% RSLogix 500 project INTRO TO PLC JOB 23 GREG.RSS, saved by version 10.00.00.00 %
PROJECT "UNTITLED"    % processor: Bul.1763 MicroLogix 1100 Series B %

PROGRAM FILES
  LAD 2   25 rungs

DATA FILES
  O0 OUTPUT  4 elements
  I1 INPUT  6 elements
  S2 STATUS  66 elements
  B3 BINARY  1 elements
  T4 TIMER  5 elements
  C5 COUNTER  8 elements
  R6 CONTROL  1 elements
  N7 INTEGER  1 elements
  F8 FLOAT  1 elements

LADDER 2
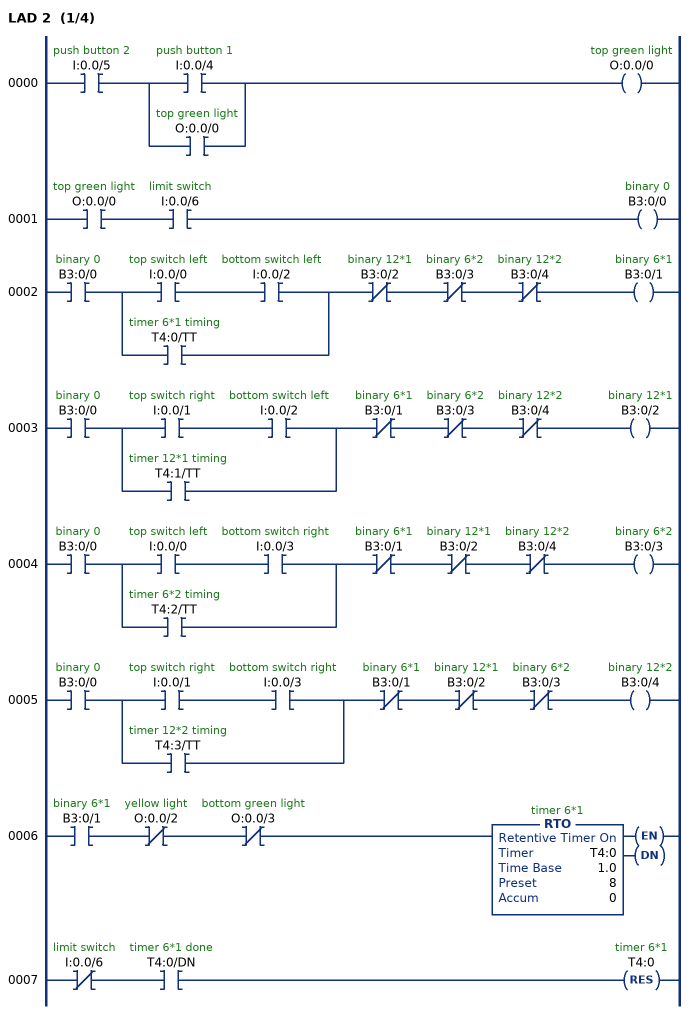
% Rung: 0 %
SOR XIC I:0.0/5 BST XIC I:0.0/4 NXB XIC O:0.0/0 BND OTE O:0.0/0 EOR
%   I:0.0/5  "push button 2" %
%   I:0.0/4  "push button 1" %
%   O:0.0/0  "top green light" %
% Rung: 1 %
SOR XIC O:0.0/0 XIC I:0.0/6 OTE B3:0/0 EOR
%   O:0.0/0  "top green light" %
%   I:0.0/6  "limit switch" %
%   B3:0/0  "binary 0" %
% Rung: 2 %
SOR XIC B3:0/0 BST XIC I:0.0/0 XIC I:0.0/2 NXB XIC T4:0/TT BND XIO B3:0/2 XIO B3:0/3 XIO B3:0/4 OTE B3:0/1 EOR
%   B3:0/0  "binary 0" %
%   I:0.0/0  "top switch left" %
%   I:0.0/2  "bottom switch left" %
%   T4:0/TT  "timer 6*1 timing" %
%   B3:0/2  "binary 12*1" %
%   B3:0/3  "binary 6*2" %
%   B3:0/4  "binary 12*2" %
%   B3:0/1  "binary 6*1" %
% Rung: 3 %
SOR XIC B3:0/0 BST XIC I:0.0/1 XIC I:0.0/2 NXB XIC T4:1/TT BND XIO B3:0/1 XIO B3:0/3 XIO B3:0/4 OTE B3:0/2 EOR
%   B3:0/0  "binary 0" %
%   I:0.0/1  "top switch right" %
%   I:0.0/2  "bottom switch left" %
%   T4:1/TT  "timer 12*1 timing" %
%   B3:0/1  "binary 6*1" %
%   B3:0/3  "binary 6*2" %
%   B3:0/4  "binary 12*2" %
%   B3:0/2  "binary 12*1" %
% Rung: 4 %
SOR XIC B3:0/0 BST XIC I:0.0/0 XIC I:0.0/3 NXB XIC T4:2/TT BND XIO B3:0/1 XIO B3:0/2 XIO B3:0/4 OTE B3:0/3 EOR
%   B3:0/0  "binary 0" %
%   I:0.0/0  "top switch left" %
%   I:0.0/3  "bottom switch right" %
%   T4:2/TT  "timer 6*2 timing" %
%   B3:0/1  "binary 6*1" %
%   B3:0/2  "binary 12*1" %
%   B3:0/4  "binary 12*2" %
%   B3:0/3  "binary 6*2" %
% Rung: 5 %
SOR XIC B3:0/0 BST XIC I:0.0/1 XIC I:0.0/3 NXB XIC T4:3/TT BND XIO B3:0/1 XIO B3:0/2 XIO B3:0/3 OTE B3:0/4 EOR
%   B3:0/0  "binary 0" %
%   I:0.0/1  "top switch right" %
%   I:0.0/3  "bottom switch right" %
%   T4:3/TT  "timer 12*2 timing" %
%   B3:0/1  "binary 6*1" %
%   B3:0/2  "binary 12*1" %
%   B3:0/3  "binary 6*2" %
%   B3:0/4  "binary 12*2" %
% Rung: 6 %
SOR XIC B3:0/1 XIO O:0.0/2 XIO O:0.0/3 RTO T4:0 1.0 8 0 EOR
%   B3:0/1  "binary 6*1" %
%   O:0.0/2  "yellow light" %
%   O:0.0/3  "bottom green light" %
%   T4:0  "timer 6*1" %
% Rung: 7 %
SOR XIO I:0.0/6 XIC T4:0/DN RES T4:0 EOR
%   I:0.0/6  "limit switch" %
%   T4:0/DN  "timer 6*1 done" %
%   T4:0  "timer 6*1" %

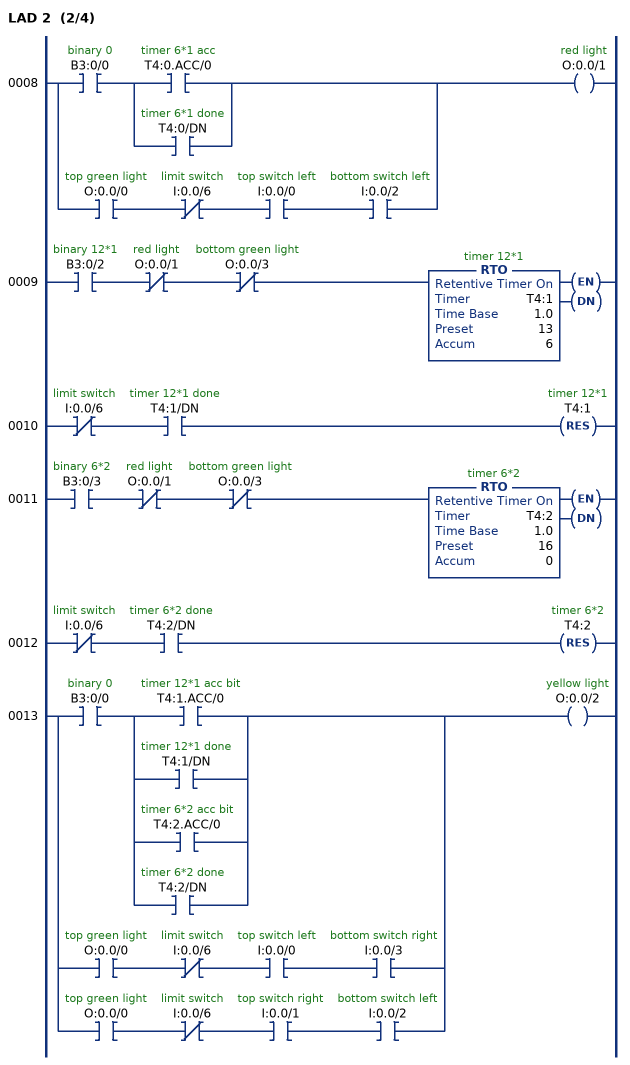
% Rung: 8 %
SOR BST XIC B3:0/0 BST XIC T4:0.ACC/0 NXB XIC T4:0/DN BND NXB XIC O:0.0/0 XIO I:0.0/6 XIC I:0.0/0 XIC I:0.0/2 BND OTE O:0.0/1 EOR
%   B3:0/0  "binary 0" %
%   T4:0.ACC/0  "timer 6*1 acc" %
%   T4:0/DN  "timer 6*1 done" %
%   O:0.0/0  "top green light" %
%   I:0.0/6  "limit switch" %
%   I:0.0/0  "top switch left" %
%   I:0.0/2  "bottom switch left" %
%   O:0.0/1  "red light" %
% Rung: 9 %
SOR XIC B3:0/2 XIO O:0.0/1 XIO O:0.0/3 RTO T4:1 1.0 13 6 EOR
%   B3:0/2  "binary 12*1" %
%   O:0.0/1  "red light" %
%   O:0.0/3  "bottom green light" %
%   T4:1  "timer 12*1" %
% Rung: 10 %
SOR XIO I:0.0/6 XIC T4:1/DN RES T4:1 EOR
%   I:0.0/6  "limit switch" %
%   T4:1/DN  "timer 12*1 done" %
%   T4:1  "timer 12*1" %
% Rung: 11 %
SOR XIC B3:0/3 XIO O:0.0/1 XIO O:0.0/3 RTO T4:2 1.0 16 0 EOR
%   B3:0/3  "binary 6*2" %
%   O:0.0/1  "red light" %
%   O:0.0/3  "bottom green light" %
%   T4:2  "timer 6*2" %
% Rung: 12 %
SOR XIO I:0.0/6 XIC T4:2/DN RES T4:2 EOR
%   I:0.0/6  "limit switch" %
%   T4:2/DN  "timer 6*2 done" %
%   T4:2  "timer 6*2" %
% Rung: 13 %
SOR BST XIC B3:0/0 BST XIC T4:1.ACC/0 NXB XIC T4:1/DN NXB XIC T4:2.ACC/0 NXB XIC T4:2/DN BND NXB XIC O:0.0/0 XIO I:0.0/6 XIC I:0.0/0 XIC I:0.0/3 NXB XIC O:0.0/0 XIO I:0.0/6 XIC I:0.0/1 XIC I:0.0/2 BND OTE O:0.0/2 EOR
%   B3:0/0  "binary 0" %
%   T4:1.ACC/0  "timer 12*1 acc bit" %
%   T4:1/DN  "timer 12*1 done" %
%   T4:2.ACC/0  "timer 6*2 acc bit" %
%   T4:2/DN  "timer 6*2 done" %
%   O:0.0/0  "top green light" %
%   I:0.0/6  "limit switch" %
%   I:0.0/0  "top switch left" %
%   I:0.0/3  "bottom switch right" %
%   I:0.0/1  "top switch right" %
%   I:0.0/2  "bottom switch left" %
%   O:0.0/2  "yellow light" %

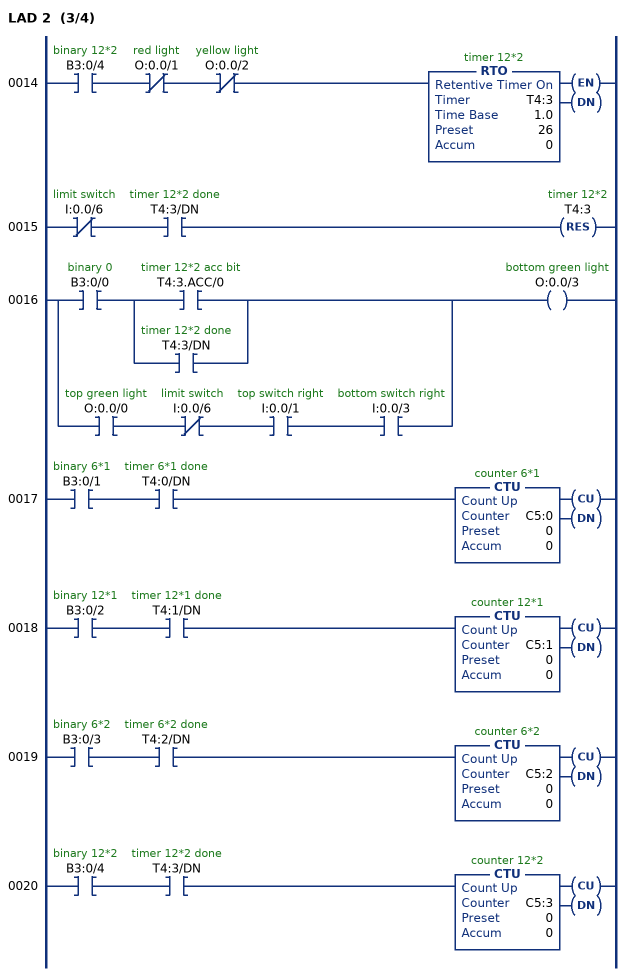
% Rung: 14 %
SOR XIC B3:0/4 XIO O:0.0/1 XIO O:0.0/2 RTO T4:3 1.0 26 0 EOR
%   B3:0/4  "binary 12*2" %
%   O:0.0/1  "red light" %
%   O:0.0/2  "yellow light" %
%   T4:3  "timer 12*2" %
% Rung: 15 %
SOR XIO I:0.0/6 XIC T4:3/DN RES T4:3 EOR
%   I:0.0/6  "limit switch" %
%   T4:3/DN  "timer 12*2 done" %
%   T4:3  "timer 12*2" %
% Rung: 16 %
SOR BST XIC B3:0/0 BST XIC T4:3.ACC/0 NXB XIC T4:3/DN BND NXB XIC O:0.0/0 XIO I:0.0/6 XIC I:0.0/1 XIC I:0.0/3 BND OTE O:0.0/3 EOR
%   B3:0/0  "binary 0" %
%   T4:3.ACC/0  "timer 12*2 acc bit" %
%   T4:3/DN  "timer 12*2 done" %
%   O:0.0/0  "top green light" %
%   I:0.0/6  "limit switch" %
%   I:0.0/1  "top switch right" %
%   I:0.0/3  "bottom switch right" %
%   O:0.0/3  "bottom green light" %
% Rung: 17 %
SOR XIC B3:0/1 XIC T4:0/DN CTU C5:0 0 0 EOR
%   B3:0/1  "binary 6*1" %
%   T4:0/DN  "timer 6*1 done" %
%   C5:0  "counter 6*1" %
% Rung: 18 %
SOR XIC B3:0/2 XIC T4:1/DN CTU C5:1 0 0 EOR
%   B3:0/2  "binary 12*1" %
%   T4:1/DN  "timer 12*1 done" %
%   C5:1  "counter 12*1" %
% Rung: 19 %
SOR XIC B3:0/3 XIC T4:2/DN CTU C5:2 0 0 EOR
%   B3:0/3  "binary 6*2" %
%   T4:2/DN  "timer 6*2 done" %
%   C5:2  "counter 6*2" %
% Rung: 20 %
SOR XIC B3:0/4 XIC T4:3/DN CTU C5:3 0 0 EOR
%   B3:0/4  "binary 12*2" %
%   T4:3/DN  "timer 12*2 done" %
%   C5:3  "counter 12*2" %

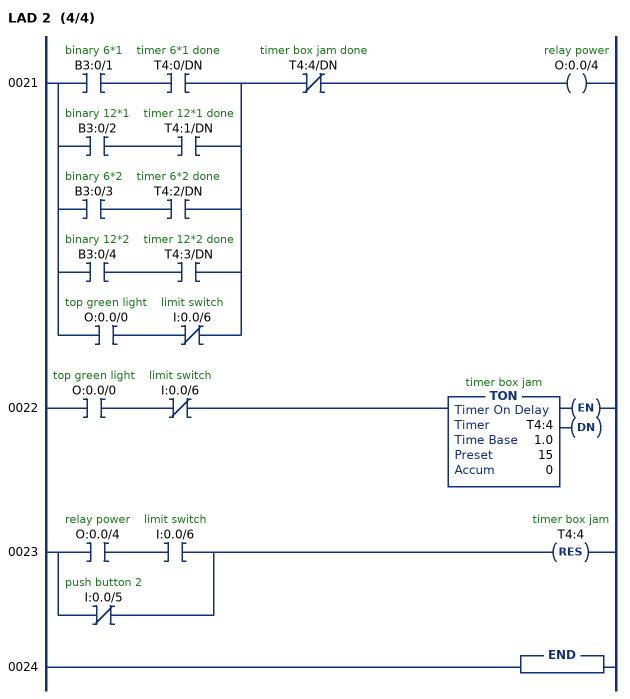
% Rung: 21 %
SOR BST BST XIC B3:0/1 XIC T4:0/DN NXB XIC B3:0/2 XIC T4:1/DN NXB XIC B3:0/3 XIC T4:2/DN NXB XIC B3:0/4 XIC T4:3/DN BND NXB XIC O:0.0/0 XIO I:0.0/6 BND XIO T4:4/DN OTE O:0.0/4 EOR
%   B3:0/1  "binary 6*1" %
%   T4:0/DN  "timer 6*1 done" %
%   B3:0/2  "binary 12*1" %
%   T4:1/DN  "timer 12*1 done" %
%   B3:0/3  "binary 6*2" %
%   T4:2/DN  "timer 6*2 done" %
%   B3:0/4  "binary 12*2" %
%   T4:3/DN  "timer 12*2 done" %
%   O:0.0/0  "top green light" %
%   I:0.0/6  "limit switch" %
%   T4:4/DN  "timer box jam done" %
%   O:0.0/4  "relay power" %
% Rung: 22 %
SOR XIC O:0.0/0 XIO I:0.0/6 TON T4:4 1.0 15 0 EOR
%   O:0.0/0  "top green light" %
%   I:0.0/6  "limit switch" %
%   T4:4  "timer box jam" %
% Rung: 23 %
SOR BST XIC O:0.0/4 XIC I:0.0/6 NXB XIO I:0.0/5 BND RES T4:4 EOR
%   O:0.0/4  "relay power" %
%   I:0.0/6  "limit switch" %
%   I:0.0/5  "push button 2" %
%   T4:4  "timer box jam" %
% Rung: 24 %
SOR END EOR

OTHER DOCUMENTED ADDRESSES
  B3:0/5  "binary green light"
  B3:0/6  "binary LL"
  C5:0.ACC/0  "timer acc"
  C5:0/CU  "counter 6*1 count up"
  C5:0/DN  "counter 6*1 done"
  C5:1.ACC/0  "counter 12*1 acc bit"
  C5:1/DN  "counter 12*1 done"
  C5:2.ACC/0  "counter 6*2 acc bit"
  C5:2/DN  "counter 6*2 done"
  C5:3.ACC/0  "counter 24*2 acc bit"
  C5:3/DN  "counter 12*2 done"
  C5:4  "counter 6*1 packs"
  C5:5  "counter 12*1 packs"
  C5:6  "counter 6*2 packs"
  C5:7  "counter 12*2 packs"
  T4:0.ACC  "timer 6*1 acc"
  T4:1.ACC  "timer 12*1 acc"
  T4:2.ACC  "timer 6*2 acc"
  T4:3.ACC  "timer 12*2 acc"
  T4:4.ACC  "timer box jam acc"

DATA TABLE (non-zero values as saved)
DATA T4
% .PRE .ACC %
% T4:0 % 8 0
% T4:1 % 13 6
% T4:2 % 16 0
% T4:3 % 26 0
% T4:4 % 15 0
